FUNCTION_BLOCK ManualCyclicCall EXTENDS Instance IMPLEMENTS I_CyclicInstance
VAR
	membership : GlobalInstanceMembership(THIS^);
	_cyclicInstanceCallback : CyclicCallback(0);
END_VAR

PROPERTY PUBLIC CyclicInstanceCallback : I_Callback
GET
CyclicInstanceCallback := _cyclicInstanceCallback;
END_GET
END_PROPERTY

METHOD PUBLIC Disable
VAR_INPUT
END_VAR
membership.Leave();
END_METHOD

METHOD PUBLIC Enable
VAR_INPUT
END_VAR
membership.Join();
END_METHOD

METHOD FB_init : BOOL
VAR_INPUT
	bInitRetains : BOOL; // if TRUE, the retain variables are initialized (warm start / cold start)
	bInCopyCode : BOOL;  // if TRUE, the instance afterwards gets moved into the copy code (online change)
	Target : I_CyclicCalled;
END_VAR
_cyclicInstanceCallback.Target := Target;
END_METHOD

END_FUNCTION_BLOCK

(* stored: Version 1.1.0.1, ProductVersion 3.1.4024.11
   POU ManualCyclicCall: Id {d2a6eae5-f4c1-4aa1-b9bb-b0e27da19250}, SpecialFunc None
   Folder Constructor: Id {95d99c90-78e5-4239-959f-5a2084f3c724}
   Property CyclicInstanceCallback: Id {b1af1ac8-3131-42cd-ae1a-263c770de573}
   Get Get: Id {3355e5d4-0172-4e55-a365-facbcd3477b6}
   Method Disable: Id {f8a54ed5-10e8-43e3-b598-39d803f73ba2}
   Method Enable: Id {03c801e5-9dd4-423c-86e3-6dcb4b0a8928}
   Method FB_init: Id {7726bab5-3c2e-47e7-b183-140b6f298cd0} *)
